{attribute 'qualified_only'}
VAR_GLOBAL
	//Output from process
	ixTram	AT %I*: BOOL;
	ixA		AT %I*: BOOL;
	ixB		AT %I*: BOOL;
	
	//Input to from Operator
	qxGotoPosB AT %Q*: BOOL;
	qxGotoPosA AT %Q*: BOOL;
	//qcStop AT %I*: BOOL;
	//qxEmergency AT %I*: BOOL;
END_VAR

(* stored: Version 1.1.0.1, ProductVersion 3.1.4024.12
   GVL GVL: Id {af0f5f45-3142-47a6-a941-102a643b77ce} *)
